(* CODESYS project tc3_hbi_cylinder.library
   Placeholder: Tc3_HBI_Cylinder
   Title: Tc3_HBI_Cylinder
   Version: 3.3.3.1
   DefaultNamespace: Tc3_HBI_Cylinder
   Company: BeckHoff SG

Project tree, tasks and I/O mapping:
  libraries: Tc2_Standard, * (Beckhoff Automation GmbH); Tc2_System, * (Beckhoff Automation GmbH); Tc2_Utilities, * (Beckhoff Automation GmbH); Tc3_HBI_System, * (BeckHoff); Tc3_System, * (Beckhoff Automation GmbH)
  04_Cylinder/
    DUTs/
      data type _ST_Cylinder
      data type _ST_Cylinder_Status
      data type ST_Cylinder
    ITFs/
      interface I_Cylinder: M_nControl, P_ipExtend, P_ipRetract, P_opExtend, P_opRetract, P_SensorDelay, P_Timeout
    POUs/
      function block FB_Cylinder [ST]: M_nControl, P_ipExtend, P_ipRetract, P_opExtend, P_opRetract, P_SensorDelay, P_sMessage, P_Timeout
  05_Vacuum/
    DUTs/
      data type _ST_Vacuum
      data type _ST_Vacuum_Status
      data type ST_Vacuum
    ITFs/
      interface I_Vacuum: M_nControl, P_ipVacuumOff, P_ipVacuumOn, P_opVacuumOff, P_opVacuumOn, P_SensorDelay, P_Timeout
    POUs/
      function block FB_Vacuum [ST]: M_nControl, P_ipVacuumOff, P_ipVacuumOn, P_opVacuumOff, P_opVacuumOn, P_SensorDelay, P_Timeout
  06_Purge/
    DUTs/
      data type _ST_Purge
      data type _ST_Purge_Status
      data type ST_Purge
    ITFs/
      interface I_Purge: M_nControl, P_ipPurgeOff, P_ipPurgeOn, P_opPurgeOff, P_opPurgeOn, P_SensorDelay, P_Timeout
    POUs/
      function block FB_Purge [ST]: M_nControl, P_ipPurgeOff, P_ipPurgeOn, P_opPurgeOff, P_opPurgeOn, P_SensorDelay, P_Timeout
  Version/
    global variables Global_Version
  Tc3_HBI_Cylinder.tmc
*)

// 04_Cylinder/DUTs/_ST_Cylinder
TYPE _ST_Cylinder EXTENDS ST_Basic :
STRUCT
	bExtend		: BOOL;
	bRetract	: BOOL;
	tTimeout	: TIME:= T#5S;
	tSensorDelay: TIME:= T#3S;
END_STRUCT
END_TYPE

// 04_Cylinder/DUTs/_ST_Cylinder_Status
TYPE _ST_Cylinder_Status EXTENDS ST_Basic_Status :
STRUCT
	ipExtend	: BOOL;
	ipRetract	: BOOL;
	opExtend	: BOOL;
	opRetract	: BOOL;
	nControl: UDINT;
END_STRUCT
END_TYPE

// 04_Cylinder/DUTs/ST_Cylinder
TYPE ST_Cylinder EXTENDS ST_Basic :
STRUCT
	bExtend		: BOOL;
	bRetract	: BOOL;
	tTimeout	: TIME:= T#5S;
	tSensorDelay: TIME:= T#3S;
	stStatus: _ST_Cylinder_Status;
END_STRUCT
END_TYPE

// 05_Vacuum/DUTs/_ST_Vacuum
TYPE _ST_Vacuum EXTENDS ST_Basic :
STRUCT
	bVacuumOn		: BOOL;
	bVacuumOff		: BOOL;
	tTimeout		: TIME:= T#5S;
	tSensorDelay	: TIME:= T#3S;
END_STRUCT
END_TYPE

// 05_Vacuum/DUTs/_ST_Vacuum_Status
TYPE _ST_Vacuum_Status EXTENDS ST_Basic_Status :
STRUCT
	ipVacuumOn		: BOOL;
	ipVacuumOff		: BOOL;
	opVacuumOn		: BOOL;
	opVacuumOff		: BOOL;
	nControl: UDINT;
END_STRUCT
END_TYPE

// 05_Vacuum/DUTs/ST_Vacuum
TYPE ST_Vacuum EXTENDS ST_Basic :
STRUCT
	bVacuumOn		: BOOL;
	bVacuumOff		: BOOL;
	tTimeout		: TIME:= T#5S;
	tSensorDelay	: TIME:= T#3S;
	stStatus: _ST_Vacuum_Status;
END_STRUCT
END_TYPE

// 06_Purge/DUTs/_ST_Purge
TYPE _ST_Purge EXTENDS ST_Basic :
STRUCT
	bPurgeOn		: BOOL;
	bPurgeOff		: BOOL;
	tTimeout		: TIME:= T#5S;
	tSensorDelay	: TIME:= T#3S;
END_STRUCT
END_TYPE

// 06_Purge/DUTs/_ST_Purge_Status
TYPE _ST_Purge_Status EXTENDS ST_Basic_Status :
STRUCT
	ipPurgeOn		: BOOL;
	ipPurgeOff		: BOOL;
	opPurgeOn		: BOOL;
	opPurgeOff		: BOOL;
	nControl: UDINT;
END_STRUCT
END_TYPE

// 06_Purge/DUTs/ST_Purge
TYPE ST_Purge EXTENDS ST_Basic :
STRUCT
	bPurgeOn		: BOOL;
	bPurgeOff		: BOOL;
	tTimeout		: TIME:= T#5S;
	tSensorDelay	: TIME:= T#3S;
	stStatus: _ST_Purge_Status;
END_STRUCT
END_TYPE

// Version/Global_Version
{attribute 'TcGenerated'}
// This function has been automatically generated from the project information.
VAR_GLOBAL CONSTANT
	{attribute 'const_non_replaced'}
	{attribute 'linkalways'}
	stLibVersion_Tc3_HBI_Cylinder : ST_LibVersion := (iMajor := 3, iMinor := 3, iBuild := 3, iRevision := 1, sVersion := '3.3.3.1');
END_VAR

// 04_Cylinder/ITFs/I_Cylinder
INTERFACE I_Cylinder EXTENDS Tc3_HBI_System.I_Basic

METHOD PUBLIC M_nControl : UDINT
VAR_INPUT
	bRetract		: BOOL;
	bExtend			: BOOL;
END_VAR
END_METHOD

PROPERTY P_ipExtend : BOOL
GET
END_GET
SET
END_SET
END_PROPERTY

PROPERTY P_ipRetract : BOOL
GET
END_GET
SET
END_SET
END_PROPERTY

PROPERTY P_opExtend : BOOL
GET
END_GET
SET
END_SET
END_PROPERTY

PROPERTY P_opRetract : BOOL
GET
END_GET
SET
END_SET
END_PROPERTY

PROPERTY P_SensorDelay : TIME
SET
END_SET
END_PROPERTY

PROPERTY P_Timeout : TIME
SET
END_SET
END_PROPERTY

END_INTERFACE

// 04_Cylinder/POUs/FB_Cylinder
//------------------------------------------------------------------------------------------
//                                                                                        	
//***************************** Beckhoff TwinCAT Examples **********************************
//                                                                                        	
//************************************* WARNING ********************************************
// This program is only an example. If it is used as a control program in any real        	
// application, Beckhoff is not responsible for any malfunction, loss or damage           	
// which could arise by using this program!                                               	
//                                                                                        	
//*************************************  Program Info. *************************************
//                                                                                        	
// PLC program name:       	FB_Cylinder (FB)                                          	
// Hardware platform:      	TwinCat PTP v3.1.4022				                          	                                  	
//                                                                                        	
// ======================================================================================== 
//         Version       Date                        Remarks                              	
// ======================================================================================== 
//         3.1.1.1      01 March 2018                First release of this example  
//         3.1.1.2      05 March 2018                Next release of this example  
//         3.2.1.1      09 March 2018                Next release of this example  
//         3.2.2.0      09 April 2018                Next release of this example 
//         3.2.2.1      13 April 2018                Next release of this example    
// ======================================================================================== 
//                                                                                        	
//******************************* Aims OF this PLC PROGRAM *********************************
//                                                                                        	
// 	3.2.2.0 added message for cylinder alarm					 			                                      	
//	3.2.2.1 sloved the cylinder timer start when alarm reset always trigger															                      	
//  3.3.3.1 add property for get set to send status out                                                                                     	
//----------------------------------------------------------------------------------------- 
FUNCTION_BLOCK FB_Cylinder EXTENDS FB_Basic IMPLEMENTS I_Cylinder
VAR	
	FB_Cylinder_M_nControl_iState	: INT;
	
	FB_Cylinder_M_nControl_bExtend		: BOOL;
	FB_Cylinder_M_nControl_bRetract		: BOOL;
	FB_Cylinder_M_nControl_ipExtend		: BOOL;
	FB_Cylinder_M_nControl_ipRetract	: BOOL;
	FB_Cylinder_M_nControl_opExtend		: BOOL;
	FB_Cylinder_M_nControl_opRetract	: BOOL;
	FB_Cylinder_M_nControl_tTimeout		: TIME:= T#5S;
	FB_Cylinder_M_nControl_tSensorDelay	: TIME:= T#3S;
	FB_Cylinder_M_nControl_sMessage		: STRING(80);
	
	FB_Cylinder_M_nControl_fbExtend_R_TRIG: Tc2_Standard.R_TRIG;
	FB_Cylinder_M_nControl_fbRetract_R_TRIG: Tc2_Standard.R_TRIG;
	
	FB_Cylinder_M_nControl_fbTimeout: Tc2_Standard.TON;
	FB_Cylinder_M_nControl_fbSensorDelay: Tc2_Standard.TON;
END_VAR

// =========================================================
	

// =========================================================

//	The result of the method is an unsigned double integer
//	0 = idle 
//	1 = coupled
//	2 = starting
//	3 = running
//	4 = aborted
// 	5 = no hardware connected
// 	6 = Spare
//	7 = pointer or index error
//	8 = mapping error
//	9 = parameter error
//	10 = complete
//	21 = cylinder extend error
// 	22 = cylinder retract error
// 	23 = vacuum on error
// 	24 = vacuum off error
// 	25 = purge on error
// 	26 = purge off error
//	Any other number = ErrorID
METHOD PUBLIC M_nControl : UDINT
VAR_INPUT	
	bRetract	: BOOL;
	bExtend		: BOOL;
END_VAR
VAR_OUTPUT
END_VAR
// =========================================================
		// Local variables
FB_Cylinder_M_nControl_bExtend:= bExtend;		
FB_Cylinder_M_nControl_bRetract:= bRetract;

// =========================================================		
		// Reset
IF _bReset THEN
	IF _bError THEN;
		FB_Cylinder_M_nControl_sMessage:= '';
		IF FB_Cylinder_M_nControl_bExtend OR FB_Cylinder_M_nControl_bRetract THEN
			FB_Cylinder_M_nControl_iState:= 01;
			ELSE FB_Cylinder_M_nControl_iState:= 00;
		END_IF
	END_IF	
END_IF

// =========================================================
		// Retract or extend position requested
	FB_Cylinder_M_nControl_fbExtend_R_TRIG(CLK:= FB_Cylinder_M_nControl_bExtend, Q=> );
	FB_Cylinder_M_nControl_fbRetract_R_TRIG(CLK:= FB_Cylinder_M_nControl_bRetract, Q=> );
	
	IF FB_Cylinder_M_nControl_fbExtend_R_TRIG.Q OR FB_Cylinder_M_nControl_fbRetract_R_TRIG.Q THEN
		FB_Cylinder_M_nControl_iState:= 01;
	END_IF
		
// =========================================================
		// Cylinder state
		
CASE FB_Cylinder_M_nControl_iState OF 
	
	00: // Do nothing
		M_nControl:= Tc3_HBI_System.cIDLE;
	01:// Reset timer
		M_nControl:= Tc3_HBI_System.cRUNNING;
		FB_Cylinder_M_nControl_fbTimeout(IN:= FALSE, PT:= FB_Cylinder_M_nControl_tTimeout, Q=> , ET=> );
		FB_Cylinder_M_nControl_fbSensorDelay(IN:= FALSE, PT:= FB_Cylinder_M_nControl_tSensorDelay, Q=> , ET=> );
		
		FB_Cylinder_M_nControl_iState:= FB_Cylinder_M_nControl_iState+1;
		
	02:// Starting
		M_nControl:= Tc3_HBI_System.cSTARTING;
		IF _bReset THEN
			FB_Cylinder_M_nControl_iState:= FB_Cylinder_M_nControl_iState-1;
			ELSIF FB_Cylinder_M_nControl_bExtend THEN
				FB_Cylinder_M_nControl_iState:= 10;
				ELSIF FB_Cylinder_M_nControl_bRetract THEN
					FB_Cylinder_M_nControl_iState:= 20;					
						ELSE FB_Cylinder_M_nControl_iState:= 00;
		END_IF
	
	10: // Extend 
		M_nControl:= Tc3_HBI_System.cRUNNING;
		FB_Cylinder_M_nControl_opRetract:= FALSE;
		FB_Cylinder_M_nControl_opExtend:= TRUE;	
		FB_Cylinder_M_nControl_fbTimeout(IN:= TRUE, PT:= FB_Cylinder_M_nControl_tTimeout, Q=> , ET=> );
		FB_Cylinder_M_nControl_fbSensorDelay(IN:= FB_Cylinder_M_nControl_ipExtend, PT:= FB_Cylinder_M_nControl_tSensorDelay, Q=> , ET=> );
		
		IF FB_Cylinder_M_nControl_fbSensorDelay.Q THEN
			FB_Cylinder_M_nControl_iState:= FB_Cylinder_M_nControl_iState+1;
			ELSE 
				IF FB_Cylinder_M_nControl_fbTimeout.Q THEN
					M_nError(nErrorID:= 21);
					FB_Cylinder_M_nControl_sMessage:= 'Cylinder extend error';
					FB_Cylinder_M_nControl_iState:= 99;
				END_IF
		END_IF
	
	11: // Extend done
		M_nControl:= Tc3_HBI_System.cCOMPLETE;
		
		IF NOT FB_Cylinder_M_nControl_bExtend THEN
			FB_Cylinder_M_nControl_iState:= 00;
		END_IF
		
	20: // Retract
		M_nControl:= Tc3_HBI_System.cRUNNING;
		FB_Cylinder_M_nControl_opExtend:= FALSE;
		FB_Cylinder_M_nControl_opRetract:= TRUE;
		FB_Cylinder_M_nControl_fbTimeout(IN:= TRUE, PT:= FB_Cylinder_M_nControl_tTimeout, Q=> , ET=> );
		FB_Cylinder_M_nControl_fbSensorDelay(IN:= FB_Cylinder_M_nControl_ipRetract, PT:= FB_Cylinder_M_nControl_tSensorDelay, Q=> , ET=> );
		
		IF FB_Cylinder_M_nControl_fbSensorDelay.Q THEN
			FB_Cylinder_M_nControl_iState:= FB_Cylinder_M_nControl_iState+1;
			ELSE 
				IF FB_Cylinder_M_nControl_fbTimeout.Q THEN
					M_nError(nErrorID:= 22);
					FB_Cylinder_M_nControl_sMessage:= 'Cylinder retract error';
					FB_Cylinder_M_nControl_iState:= 99;
				END_IF
		END_IF
		
	21: // Retract done
		M_nControl:= Tc3_HBI_System.cCOMPLETE;
		
		IF NOT FB_Cylinder_M_nControl_bRetract THEN
			FB_Cylinder_M_nControl_iState:= 0;
		END_IF
		
	99: // Error state
		M_nControl:= Tc3_HBI_System.cABORTED;
		
		FB_Cylinder_M_nControl_fbSensorDelay(IN:= FALSE, PT:= T#0S, Q=> , ET=> );
		FB_Cylinder_M_nControl_fbTimeout(IN:= FALSE, PT:= T#0S, Q=> , ET=> );
		IF NOT FB_Cylinder_M_nControl_bExtend AND NOT FB_Cylinder_M_nControl_bRetract THEN
			FB_Cylinder_M_nControl_iState:= 0;
		END_IF

ELSE
	FB_Cylinder_M_nControl_iState:= 0;
END_CASE
// =========================================================
END_METHOD

{warning 'add property implementation'}
PROPERTY P_ipExtend : BOOL
GET
P_ipExtend:= FB_Cylinder_M_nControl_ipExtend;
END_GET
SET
FB_Cylinder_M_nControl_ipExtend := P_ipExtend;
END_SET
END_PROPERTY

{warning 'add property implementation'}
PROPERTY P_ipRetract : BOOL
GET
P_ipRetract:= FB_Cylinder_M_nControl_ipRetract;
END_GET
SET
FB_Cylinder_M_nControl_ipRetract := P_ipRetract;
END_SET
END_PROPERTY

{warning 'add property implementation'}
PROPERTY P_opExtend : BOOL
GET
P_opExtend := FB_Cylinder_M_nControl_opExtend;
END_GET
SET
FB_Cylinder_M_nControl_opExtend:= P_opExtend;
END_SET
END_PROPERTY

{warning 'add property implementation'}
PROPERTY P_opRetract : BOOL
GET
P_opRetract := FB_Cylinder_M_nControl_opRetract;
END_GET
SET
FB_Cylinder_M_nControl_opRetract:= P_opRetract;
END_SET
END_PROPERTY

PROPERTY P_SensorDelay : TIME
SET
FB_Cylinder_M_nControl_tSensorDelay:= P_SensorDelay;
END_SET
END_PROPERTY

PROPERTY PUBLIC P_sMessage : string
GET
P_sMessage:= FB_Cylinder_M_nControl_sMessage;
END_GET
END_PROPERTY

{warning 'add property implementation'}
PROPERTY P_Timeout : TIME
SET
FB_Cylinder_M_nControl_tTimeout:= P_Timeout;
END_SET
END_PROPERTY

END_FUNCTION_BLOCK

// 05_Vacuum/ITFs/I_Vacuum
INTERFACE I_Vacuum EXTENDS Tc3_HBI_System.I_Basic

METHOD M_nControl : UDINT
VAR_INPUT
	bVacuumOff		: BOOL;
	bVacuumOn		: BOOL;
END_VAR
END_METHOD

PROPERTY P_ipVacuumOff : BOOL
GET
END_GET
SET
END_SET
END_PROPERTY

PROPERTY P_ipVacuumOn : BOOL
GET
END_GET
SET
END_SET
END_PROPERTY

PROPERTY P_opVacuumOff : BOOL
GET
END_GET
SET
END_SET
END_PROPERTY

PROPERTY P_opVacuumOn : BOOL
GET
END_GET
SET
END_SET
END_PROPERTY

PROPERTY P_SensorDelay : TIME
SET
END_SET
END_PROPERTY

PROPERTY P_Timeout : TIME
SET
END_SET
END_PROPERTY

END_INTERFACE

// 05_Vacuum/POUs/FB_Vacuum
//------------------------------------------------------------------------------------------
//                                                                                        	
//***************************** Beckhoff TwinCAT Examples **********************************
//                                                                                        	
//************************************* WARNING ********************************************
// This program is only an example. If it is used as a control program in any real        	
// application, Beckhoff is not responsible for any malfunction, loss or damage           	
// which could arise by using this program!                                               	
//                                                                                        	
//*************************************  Program Info. *************************************
//                                                                                        	
// PLC program name:       	FB_Vacuum (FB)                                          	
// Hardware platform:      	TwinCat PTP v3.1.4022				                          	                                  	
//                                                                                        	
// ======================================================================================== 
//         Version       Date                        Remarks                              	
// ======================================================================================== 
//         3.1.1.1      01 March 2018                First release of this example 
//         3.1.1.2      05 March 2018                Next release of this example    
//         3.2.1.1      09 March 2018                Next release of this example 
//         3.3.1.1      09 March 2018                Next release of this example  
// ======================================================================================== 
//                                                                                        	
//******************************* Aims OF this PLC PROGRAM *********************************
//                                                                                        	
// 	3.2.2.0 added message for vacuum alarm 						 			                                      	
//																	                      	
//                                                                                        	
//----------------------------------------------------------------------------------------- 
FUNCTION_BLOCK FB_Vacuum EXTENDS FB_Basic IMPLEMENTS I_Vacuum
VAR 
	FB_Vacuum_M_nControl_iState	: INT;
	
	FB_Vacuum_M_nControl_bVacuumOn		: BOOL;
	FB_Vacuum_M_nControl_bVacuumOff		: BOOL;
	FB_Vacuum_M_nControl_ipVacuumOn		: BOOL;
	FB_Vacuum_M_nControl_ipVacuumOff	: BOOL;
	FB_Vacuum_M_nControl_opVacuumOn		: BOOL;
	FB_Vacuum_M_nControl_opVacuumOff	: BOOL;
	FB_Vacuum_M_nControl_tTimeout		: TIME:= T#5S;
	FB_Vacuum_M_nControl_tSensorDelay	: TIME:= T#3S;
	FB_Vacuum_M_nControl_sMessage		: STRING(80);
	
	FB_Vacuum_M_nControl_fbVacuumOn_R_TRIG: Tc2_Standard.R_TRIG;
	FB_Vacuum_M_nControl_fbVacuumOff_R_TRIG: Tc2_Standard.R_TRIG;
	
	FB_Vacuum_M_nControl_fbTimeout: Tc2_Standard.TON;
	FB_Vacuum_M_nControl_fbSensorDelay: Tc2_Standard.TON;
END_VAR

//	The result of the method is an unsigned double integer
//	0 = idle 
//	1 = coupled
//	2 = starting
//	3 = running
//	4 = aborted
// 	5 = no hardware connected
// 	6 = Spare
//	7 = pointer or index error
//	8 = mapping error
//	9 = parameter error
//	10 = complete
//	21 = cylinder extend error
// 	22 = cylinder retract error
// 	23 = vacuum on error
// 	24 = vacuum off error
// 	25 = purge on error
// 	26 = purge off error
//	Any other number = ErrorID
METHOD PUBLIC M_nControl : UDINT
VAR_INPUT	
	bVacuumOff		: BOOL;
	bVacuumOn		: BOOL;
END_VAR
// =========================================================
		// Local variables
FB_Vacuum_M_nControl_bVacuumOn:= bVacuumOn;		
FB_Vacuum_M_nControl_bVacuumOff:= bVacuumOff;

// =========================================================		
		// Reset
IF _bReset THEN
	IF _bError THEN;
		FB_Vacuum_M_nControl_sMessage:= '';
		IF FB_Vacuum_M_nControl_bVacuumOn OR FB_Vacuum_M_nControl_bVacuumOff THEN
			FB_Vacuum_M_nControl_iState:= 01;
			ELSE FB_Vacuum_M_nControl_iState:= 00;
		END_IF
	END_IF	
END_IF

// =========================================================
		// Vacuum off or on requested
	FB_Vacuum_M_nControl_fbVacuumOn_R_TRIG(CLK:= FB_Vacuum_M_nControl_bVacuumOn, Q=> );
	FB_Vacuum_M_nControl_fbVacuumOff_R_TRIG(CLK:= FB_Vacuum_M_nControl_bVacuumOff, Q=> );
	
	IF FB_Vacuum_M_nControl_fbVacuumOn_R_TRIG.Q OR FB_Vacuum_M_nControl_fbVacuumOff_R_TRIG.Q THEN
		FB_Vacuum_M_nControl_iState:= 01;
	END_IF
		
// =========================================================
		// Vacuum state
		
CASE FB_Vacuum_M_nControl_iState OF 
	
	00: // Do nothing
		M_nControl:= Tc3_HBI_System.cIDLE;
		
	01:// Reset timer
		M_nControl:= Tc3_HBI_System.cRUNNING;
		FB_Vacuum_M_nControl_fbTimeout(IN:= FALSE, PT:= FB_Vacuum_M_nControl_tTimeout, Q=> , ET=> );
		FB_Vacuum_M_nControl_fbSensorDelay(IN:= FALSE, PT:= FB_Vacuum_M_nControl_tSensorDelay, Q=> , ET=> );
		
		FB_Vacuum_M_nControl_iState:= FB_Vacuum_M_nControl_iState+1;
		
	02:// Starting
		M_nControl:= Tc3_HBI_System.cSTARTING;
		IF _bReset THEN
			FB_Vacuum_M_nControl_iState:= FB_Vacuum_M_nControl_iState-1;
			ELSIF FB_Vacuum_M_nControl_bVacuumOn THEN
				FB_Vacuum_M_nControl_iState:= 10;
				ELSIF FB_Vacuum_M_nControl_bVacuumOff THEN
					FB_Vacuum_M_nControl_iState:= 20;
					ELSE FB_Vacuum_M_nControl_iState:= 00;
		END_IF
	
	10: // Vacuum on
		M_nControl:= Tc3_HBI_System.cRUNNING;
		FB_Vacuum_M_nControl_opVacuumOff:= FALSE;
		FB_Vacuum_M_nControl_opVacuumOn:= TRUE;	
		FB_Vacuum_M_nControl_fbTimeout(IN:= TRUE, PT:= FB_Vacuum_M_nControl_tTimeout, Q=> , ET=> );
		FB_Vacuum_M_nControl_fbSensorDelay(IN:= FB_Vacuum_M_nControl_ipVacuumOn, PT:= FB_Vacuum_M_nControl_tSensorDelay, Q=> , ET=> );
		
		IF FB_Vacuum_M_nControl_fbSensorDelay.Q THEN
			FB_Vacuum_M_nControl_iState:= FB_Vacuum_M_nControl_iState+1;
			ELSE 
				IF FB_Vacuum_M_nControl_fbTimeout.Q THEN
					M_nError(nErrorID:= 23);
					M_nControl:= 23;
					FB_Vacuum_M_nControl_sMessage:= 'Vacuum on error';
				END_IF
		END_IF
	
	11: // Vacuum done
		M_nControl:= Tc3_HBI_System.cCOMPLETE;
		
		IF NOT FB_Vacuum_M_nControl_bVacuumOn THEN
			FB_Vacuum_M_nControl_iState:= 00;
		END_IF
		
	20: // Vacuum off
		M_nControl:= Tc3_HBI_System.cRUNNING;
		FB_Vacuum_M_nControl_opVacuumOn:= FALSE;
		FB_Vacuum_M_nControl_opVacuumOff:= TRUE;
		FB_Vacuum_M_nControl_fbTimeout(IN:= TRUE, PT:= FB_Vacuum_M_nControl_tTimeout, Q=> , ET=> );
		FB_Vacuum_M_nControl_fbSensorDelay(IN:= FB_Vacuum_M_nControl_ipVacuumOff, PT:= FB_Vacuum_M_nControl_tSensorDelay, Q=> , ET=> );
		
		IF FB_Vacuum_M_nControl_fbSensorDelay.Q THEN
			FB_Vacuum_M_nControl_iState:= FB_Vacuum_M_nControl_iState+1;
			ELSE 
				IF FB_Vacuum_M_nControl_fbTimeout.Q THEN
					M_nError(nErrorID:= 24);
					M_nControl:= 24;
					FB_vacuum_M_nControl_sMessage:= 'Vacuum off error';
				END_IF
		END_IF
		
	21: // Vacuum done
		M_nControl:= Tc3_HBI_System.cCOMPLETE;
		
		IF NOT FB_Vacuum_M_nControl_bVacuumOff THEN
			FB_Vacuum_M_nControl_iState:= 0;
		END_IF
		
	99: // Error state
		M_nControl:= Tc3_HBI_System.cABORTED;
		FB_Vacuum_M_nControl_fbTimeout(IN:= FALSE, PT:= T#0S, Q=> , ET=> );
		FB_Vacuum_M_nControl_fbSensorDelay(IN:= FALSE, PT:= T#0S, Q=> , ET=> );
		
		IF NOT FB_Vacuum_M_nControl_bVacuumOn AND NOT FB_Vacuum_M_nControl_bVacuumOff THEN
			FB_Vacuum_M_nControl_iState:= 0;
		END_IF
ELSE
	FB_Vacuum_M_nControl_iState:= 00;
	
END_CASE
// =========================================================
END_METHOD

{warning 'add property implementation'}
PROPERTY P_ipVacuumOff : BOOL
GET
P_ipVacuumOff:= FB_Vacuum_M_nControl_ipVacuumOff
END_GET
SET
FB_Vacuum_M_nControl_ipVacuumOff := P_ipVacuumOff;
END_SET
END_PROPERTY

{warning 'add property implementation'}
PROPERTY P_ipVacuumOn : BOOL
GET
P_ipVacuumOn:= FB_Vacuum_M_nControl_ipVacuumOn
END_GET
SET
FB_Vacuum_M_nControl_ipVacuumOn := P_ipVacuumOn;
END_SET
END_PROPERTY

{warning 'add property implementation'}
PROPERTY P_opVacuumOff : BOOL
GET
P_opVacuumOff := FB_Vacuum_M_nControl_bVacuumOff;
END_GET
SET
FB_Vacuum_M_nControl_bVacuumOff:= P_opVacuumOff;
END_SET
END_PROPERTY

{warning 'add property implementation'}
PROPERTY P_opVacuumOn : BOOL
GET
P_opVacuumOn := FB_Vacuum_M_nControl_bVacuumOn;
END_GET
SET
FB_Vacuum_M_nControl_bVacuumOn:= P_opVacuumOn
END_SET
END_PROPERTY

PROPERTY P_SensorDelay : TIME
SET
FB_Vacuum_M_nControl_tSensorDelay:= P_SensorDelay;
END_SET
END_PROPERTY

PROPERTY P_Timeout : TIME
SET
FB_Vacuum_M_nControl_tTimeout:= P_Timeout;
END_SET
END_PROPERTY

END_FUNCTION_BLOCK

// 06_Purge/ITFs/I_Purge
INTERFACE I_Purge EXTENDS Tc3_HBI_System.I_Basic

METHOD M_nControl : UDINT
VAR_INPUT
	bPurgeOn	: BOOL;
	bPurgeOff	: BOOL;
END_VAR
END_METHOD

PROPERTY P_ipPurgeOff : BOOL
GET
END_GET
SET
END_SET
END_PROPERTY

PROPERTY P_ipPurgeOn : BOOL
GET
END_GET
SET
END_SET
END_PROPERTY

PROPERTY P_opPurgeOff : BOOL
GET
END_GET
SET
END_SET
END_PROPERTY

PROPERTY P_opPurgeOn : BOOL
GET
END_GET
SET
END_SET
END_PROPERTY

PROPERTY P_SensorDelay : TIME
SET
END_SET
END_PROPERTY

PROPERTY P_Timeout : TIME
SET
END_SET
END_PROPERTY

END_INTERFACE

// 06_Purge/POUs/FB_Purge
//------------------------------------------------------------------------------------------
//                                                                                        	
//***************************** Beckhoff TwinCAT Examples **********************************
//                                                                                        	
//************************************* WARNING ********************************************
// This program is only an example. If it is used as a control program in any real        	
// application, Beckhoff is not responsible for any malfunction, loss or damage           	
// which could arise by using this program!                                               	
//                                                                                        	
//*************************************  Program Info. *************************************
//                                                                                        	
// PLC program name:       	FB_Purge (FB)                                          	
// Hardware platform:      	TwinCat PTP v3.1.4022				                          	                                  	
//                                                                                        	
// ======================================================================================== 
//         Version       Date                        Remarks                              	
// ======================================================================================== 
//         3.1.1.1      01 March 2018                First release of this example 
//         3.1.1.2      05 March 2018                Next release of this example 
//         3.1.2.1      06 March 2018                Remove purge auto off 
//         3.2.1.1      09 March 2018                Next release of this example   
// ======================================================================================== 
//                                                                                        	
//******************************* Aims OF this PLC PROGRAM *********************************
// 	3.3.1.1 added message for purge alarm                                                                                       	
// 									 			                                      	
//																	                      	
//                                                                                        	
//----------------------------------------------------------------------------------------- 
FUNCTION_BLOCK FB_Purge EXTENDS FB_Basic IMPLEMENTS I_Purge
VAR 
	FB_Purge_M_nControl_iState	: INT;
	
	FB_Purge_M_nControl_bPurgeOn		: BOOL;
	FB_Purge_M_nControl_bPurgeOff		: BOOL;
	FB_Purge_M_nControl_ipPurgeOn		: BOOL;
	FB_Purge_M_nControl_ipPurgeOff		: BOOL;
	FB_Purge_M_nControl_opPurgeOn		: BOOL;
	FB_Purge_M_nControl_opPurgeOff		: BOOL;
	FB_Purge_M_nControl_tTimeout		: TIME:= T#5S;
	FB_Purge_M_nControl_tSensorDelay	: TIME:= T#3S;
	FB_Purge_M_nControl_sMessage		: STRING(80);
	
	FB_Purge_M_nControl_fbPurgeOn_R_TRIG: Tc2_Standard.R_TRIG;
	FB_Purge_M_nControl_fbPurgeOff_R_TRIG: Tc2_Standard.R_TRIG;
	
	FB_Purge_M_nControl_fbTimeout: Tc2_Standard.TON;
	FB_Purge_M_nControl_fbSensorDelay: Tc2_Standard.TON;
END_VAR

// =========================================================
	
// =========================================================

//	The result of the method is an unsigned double integer
//	0 = idle 
//	1 = coupled
//	2 = starting
//	3 = running
//	4 = aborted
// 	5 = no hardware connected
// 	6 = Spare
//	7 = pointer or index error
//	8 = mapping error
//	9 = parameter error
//	10 = complete
//	21 = cylinder extend error
// 	22 = cylinder retract error
// 	23 = vacuum on error
// 	24 = vacuum off error
// 	25 = purge on error
// 	26 = purge off error
//	Any other number = ErrorID
METHOD PUBLIC M_nControl : UDINT
VAR_INPUT	
	bPurgeOn		: BOOL;
	bPurgeOff		: BOOL;
END_VAR
// =========================================================
		// Local variables
FB_Purge_M_nControl_bPurgeOn:= bPurgeOn;		
FB_Purge_M_nControl_bPurgeOff:= bPurgeoff;

// =========================================================		
		// Reset
IF _bReset THEN
	IF _bError THEN;
		FB_Purge_M_nControl_sMessage:= '';
		IF FB_Purge_M_nControl_bPurgeOn OR FB_Purge_M_nControl_bPurgeOff THEN
			FB_Purge_M_nControl_iState:= 01;
			ELSE FB_Purge_M_nControl_iState:= 00;
		END_IF
	END_IF	
END_IF

// =========================================================
		// Purge off or on requested
	FB_Purge_M_nControl_fbPurgeOn_R_TRIG(CLK:= FB_Purge_M_nControl_bPurgeOn, Q=> );
	FB_Purge_M_nControl_fbPurgeOff_R_TRIG(CLK:= FB_Purge_M_nControl_bPurgeOff, Q=> );
	
	IF FB_Purge_M_nControl_fbPurgeOn_R_TRIG.Q OR FB_Purge_M_nControl_fbPurgeOff_R_TRIG.Q THEN
		FB_Purge_M_nControl_iState:= 01;
	END_IF
		
// =========================================================
		// Purge state
		
CASE FB_Purge_M_nControl_iState OF 
	
	00: // Do nothing
		M_nControl:= Tc3_HBI_System.cIDLE;
		
	01:// Reset timer
		M_nControl:= Tc3_HBI_System.cRUNNING;
		FB_Purge_M_nControl_fbTimeout(IN:= FALSE, PT:= FB_Purge_M_nControl_tTimeout, Q=> , ET=> );
		FB_Purge_M_nControl_fbSensorDelay(IN:= FALSE, PT:= FB_Purge_M_nControl_tSensorDelay, Q=> , ET=> );
		
		FB_Purge_M_nControl_iState:= FB_Purge_M_nControl_iState+1;
		
	02:// Starting
		M_nControl:= Tc3_HBI_System.cSTARTING;
		IF _bReset THEN
			FB_Purge_M_nControl_iState:= FB_Purge_M_nControl_iState-1;
			ELSIF FB_Purge_M_nControl_bPurgeOn THEN
				FB_Purge_M_nControl_iState:= 10;
				ELSIF FB_Purge_M_nControl_bPurgeOff THEN
					FB_Purge_M_nControl_iState:= 20;
					ELSE FB_Purge_M_nControl_iState:= 00;
		END_IF
	
	10: // Purge on
		M_nControl:= Tc3_HBI_System.cRUNNING;
		FB_Purge_M_nControl_opPurgeOff:= FALSE;
		FB_Purge_M_nControl_opPurgeOn:= TRUE;	
		FB_Purge_M_nControl_fbTimeout(IN:= TRUE, PT:= FB_Purge_M_nControl_tTimeout, Q=> , ET=> );
		FB_Purge_M_nControl_fbSensorDelay(IN:= FB_Purge_M_nControl_ipPurgeOn, PT:= FB_Purge_M_nControl_tSensorDelay, Q=> , ET=> );
		
		IF FB_Purge_M_nControl_fbSensorDelay.Q THEN
			FB_Purge_M_nControl_iState:= FB_Purge_M_nControl_iState+1;
			ELSE 
				IF FB_Purge_M_nControl_fbTimeout.Q THEN
					M_nError(nErrorID:= 25);
					M_nControl:= 25;
					FB_Purge_M_nControl_sMessage:= 'Purge on error';
				END_IF
		END_IF
	
	11: // Purge done
		M_nControl:= Tc3_HBI_System.cCOMPLETE;
(*		FB_Purge_M_nControl_opPurgeOff:= FALSE;
		FB_Purge_M_nControl_opPurgeOn:= FALSE;	
*)		
		IF NOT FB_Purge_M_nControl_bPurgeOn THEN
			FB_Purge_M_nControl_iState:= 00;
		END_IF
		
	20: // purge off
		M_nControl:= Tc3_HBI_System.cRUNNING;
		FB_Purge_M_nControl_opPurgeOn:= FALSE;
		FB_Purge_M_nControl_opPurgeOff:= TRUE;
		FB_Purge_M_nControl_fbTimeout(IN:= TRUE, PT:= FB_Purge_M_nControl_tTimeout, Q=> , ET=> );
		FB_Purge_M_nControl_fbSensorDelay(IN:= FB_Purge_M_nControl_ipPurgeOff, PT:= FB_Purge_M_nControl_tSensorDelay, Q=> , ET=> );
		
		IF FB_Purge_M_nControl_fbSensorDelay.Q THEN
			FB_Purge_M_nControl_iState:= FB_Purge_M_nControl_iState+1;
			ELSE 
				IF FB_Purge_M_nControl_fbTimeout.Q THEN
					M_nError(nErrorID:= 26);
					M_nControl:= 26;
					FB_Purge_M_nControl_sMessage:= 'Purge off error';
				END_IF
		END_IF
		
	21: // Purge done
		M_nControl:= Tc3_HBI_System.cCOMPLETE;
(*		FB_Purge_M_nControl_opPurgeOn:= FALSE;
		FB_Purge_M_nControl_opPurgeOff:= FALSE;
*)		
		IF NOT FB_Purge_M_nControl_bPurgeOff THEN
			FB_Purge_M_nControl_iState:= 00;
		END_IF
		
	99: // Error state
		M_nControl:= Tc3_HBI_System.cABORTED;
		
		FB_Purge_M_nControl_fbTimeout(IN:= FALSE, PT:= T#0S, Q=> , ET=> );
		FB_Purge_M_nControl_fbSensorDelay(IN:= FALSE, PT:= T#0S, Q=> , ET=> );
		IF NOT FB_Purge_M_nControl_bPurgeOn AND NOT FB_Purge_M_nControl_bPurgeOff THEN
			FB_Purge_M_nControl_iState:= 00;
		END_IF
		
ELSE
	FB_Purge_M_nControl_iState:= 00;
END_CASE
// =========================================================
END_METHOD

PROPERTY PUBLIC P_ipPurgeOff : BOOL
GET
P_ipPurgeOff:= FB_Purge_M_nControl_ipPurgeOff;
END_GET
SET
FB_Purge_M_nControl_ipPurgeOff:= P_ipPurgeOff;
END_SET
END_PROPERTY

PROPERTY PUBLIC P_ipPurgeOn : BOOL
GET
P_ipPurgeOn:= FB_Purge_M_nControl_ipPurgeOn;
END_GET
SET
FB_Purge_M_nControl_ipPurgeOn:= P_ipPurgeOn;
END_SET
END_PROPERTY

{warning 'add property implementation'}
PROPERTY P_opPurgeOff : BOOL
GET
P_opPurgeOff:= FB_Purge_M_nControl_opPurgeOff;
END_GET
SET
FB_Purge_M_nControl_opPurgeOff:= P_opPurgeOff;
END_SET
END_PROPERTY

PROPERTY PUBLIC P_opPurgeOn : BOOL
GET
P_opPurgeOn:= FB_Purge_M_nControl_opPurgeOn;
END_GET
SET
FB_Purge_M_nControl_opPurgeOn:= P_opPurgeOn;
END_SET
END_PROPERTY

PROPERTY P_SensorDelay : TIME
SET
FB_Purge_M_nControl_tSensorDelay:= P_SensorDelay;
END_SET
END_PROPERTY

PROPERTY P_Timeout : TIME
SET
FB_Purge_M_nControl_tTimeout:= P_Timeout;
END_SET
END_PROPERTY

END_FUNCTION_BLOCK
